// TIA Portal V19 export
FUNCTION_BLOCK "TYPIC_C402_IF_VKL"   // FB112, FBD
TITLE = TYPIC_C402_IF_VKL: Verkeerslicht
{ S7_Optimized_Access := 'TRUE' }
AUTHOR : OCOTECH
FAMILY : Typical
NAME : C402.702
// Logisch Object Besturing: C402.702
// 
// De interne functie verkeerslicht verzorgt de interne besturing, bewaking en fysieke aansturing van een verkeerslicht.
// 
// Het verkeerslicht kan via sturingen (vanuit 3B) of via handmatige bedieningen (aanraakscherm) op volgende standen gezet worden:
//  UIT (gedoofd)
//  ROOD
//  GROEN
//  GEEL KNIPPEREN
// 
// De stand “Geel vast” kan niet via sturing of bediening gekozen worden. De stand “Geel vast” wordt door deze typical altijd automatisch toegepast als overgang naar stand “Rood”.
// stored: MemoryReserve 10, SetENOAutomatically false
   VAR_INPUT
      EXT_AUT { ExternalAccessible := 'False'; ExternalVisible := 'False'; ExternalWritable := 'False'} : Bool;   // Externe (hoofd) beveiliging (1 = OK)
      EXT_HW { ExternalAccessible := 'False'; ExternalVisible := 'False'; ExternalWritable := 'False'} : Bool;   // Sturings hardware (PLC) bewaking (1 = OK)
      HULP_KNIP { ExternalAccessible := 'False'; ExternalVisible := 'False'; ExternalWritable := 'False'} : Bool;   // Knippersignaal, x tijd Hoog, x tijd Laag
      IN_AUT_C402 { ExternalAccessible := 'False'; ExternalVisible := 'False'; ExternalWritable := 'False'} : Bool;   // Beveiligingen: serie geschakelde terugmelding (1 = OK)
      IN_ROOD { ExternalAccessible := 'False'; ExternalVisible := 'False'; ExternalWritable := 'False'} : Bool;   // Terugmelding: rood aan (stroommeting)
      IN_GEEL { ExternalAccessible := 'False'; ExternalVisible := 'False'; ExternalWritable := 'False'} : Bool;   // Terugmelding: geel aan (stroommeting)
      IN_GROE { ExternalAccessible := 'False'; ExternalVisible := 'False'; ExternalWritable := 'False'} : Bool;   // Terugmelding: groen aan (stroommeting)
      CFG_TYD_FB { ExternalAccessible := 'False'; ExternalVisible := 'False'; ExternalWritable := 'False'} : Time;   // Vertragingstijd storing terugmelding
      CFG_GEEL_TYD { ExternalAccessible := 'False'; ExternalVisible := 'False'; ExternalWritable := 'False'} : Time;   // Tijdsduur verkeerslicht geel, vooraleer naar rood
      CFG_SNEL_GEEL_TYD { ExternalAccessible := 'False'; ExternalVisible := 'False'; ExternalWritable := 'False'} : Time;   // Tijdsduur verkeerslicht geel, vooraleer naar rood, bij versneld sluiten
      CFG_TYD_ONHD { ExternalAccessible := 'False'; ExternalVisible := 'False'; ExternalWritable := 'False'} : Time;   // Tijdsduur aansturing lenzen bij automatische onderhoudstesten
   END_VAR
   VAR_OUTPUT
      VAR_IF_VKL { ExternalAccessible := 'False'; ExternalVisible := 'False'; ExternalWritable := 'False'} : "C402_VAR_IF_VKL_TYPIC";   // Struct met alle variabelen naar bovenliggende functies
      OUT_ROOD { ExternalAccessible := 'False'; ExternalVisible := 'False'; ExternalWritable := 'False'} : Bool;   // Aansturing rood
      OUT_GEEL { ExternalAccessible := 'False'; ExternalVisible := 'False'; ExternalWritable := 'False'} : Bool;   // Aansturing geel
      OUT_GROE { ExternalAccessible := 'False'; ExternalVisible := 'False'; ExternalWritable := 'False'} : Bool;   // Aansturing groen
   END_VAR
   VAR_IN_OUT
      STU_IF_VKL : "C402_STU_IF_VKL_TYPIC";   // Struct met alle sturingen naar de functie (IF) in de interne sturing van het verkeerslicht
      STU_AFS_IF_VKL : "C402_STU_AFS_IF_VKL_TYPIC";   // Struct met alle sturingen naar de functie (IF) van de verkeerslichten
   END_VAR
   VAR
      STO { ExternalWritable := 'False'} : Struct   // Storingen
         A001 { ExternalAccessible := 'False'; ExternalVisible := 'False'} : Bool;   // Beveiliging aangesproken
         AT01 { ExternalAccessible := 'False'; ExternalVisible := 'False'} : Bool;   // De rode lens is defect
         AT02 { ExternalAccessible := 'False'; ExternalVisible := 'False'} : Bool;   // De gele lens is defect
         AT03 { ExternalAccessible := 'False'; ExternalVisible := 'False'} : Bool;   // De groene lens is defect
         AT04 { ExternalAccessible := 'False'; ExternalVisible := 'False'} : Bool;   // De stand rood kan niet getoond worden
         AT05 { ExternalAccessible := 'False'; ExternalVisible := 'False'} : Bool;   // De stand geel kan niet getoond worden
         AT06 { ExternalAccessible := 'False'; ExternalVisible := 'False'} : Bool;   // De stand geel knipperen kan niet getoond worden
         AT07 { ExternalAccessible := 'False'; ExternalVisible := 'False'} : Bool;   // De stand groen kan niet getoond worden
      END_STRUCT;
      VAR { ExternalWritable := 'False'} : Struct   // Variabelen
         HAND_ROOD_SWA { ExternalAccessible := 'False'; ExternalVisible := 'False'} : Bool;   // 1 = Rood gewenst, via handbediening
         HAND_KNIP_SWA { ExternalAccessible := 'False'; ExternalVisible := 'False'} : Bool;   // 1 = Geel knipperen gewenst, via handbediening
         HAND_GROE_SWA { ExternalAccessible := 'False'; ExternalVisible := 'False'} : Bool;   // 1 = Groen gewenst, via handbediening
         ROOD_SWA { ExternalAccessible := 'False'; ExternalVisible := 'False'} : Bool;   // 1 = Rood gewenst
         KNIP_SWA { ExternalAccessible := 'False'; ExternalVisible := 'False'} : Bool;   // 1 = Geel knipperen gewenst
         GROEN_SWA { ExternalAccessible := 'False'; ExternalVisible := 'False'} : Bool;   // 1 = Groen gewenst
         ROOD_AAN_SWA { ExternalAccessible := 'False'; ExternalVisible := 'False'} : Bool;   // 1 = Rood gewenst, rode lens aansturen
         GEEL_AAN_SWA { ExternalAccessible := 'False'; ExternalVisible := 'False'} : Bool;   // 1 = Rood gewenst, gele lens aansturen
         GEEL_KNIP { ExternalAccessible := 'False'; ExternalVisible := 'False'} : Bool;   // Knippersignaal voor geel licht 1 = AAN / 0 = UIT
         STO_ROOD_AAN { ExternalAccessible := 'False'; ExternalVisible := 'False'} : Bool;   // 1 = Rode lens defect, geen terugmelding bij aansturen
         STO_ROOD_UIT { ExternalAccessible := 'False'; ExternalVisible := 'False'} : Bool;   // 1 = Rode lens defect, terugmelding aan bij afsturen
         STO_GEEL_AAN { ExternalAccessible := 'False'; ExternalVisible := 'False'} : Bool;   // 1 = Gele lens defect, geen terugmelding bij aansturen
         STO_GEEL_UIT { ExternalAccessible := 'False'; ExternalVisible := 'False'} : Bool;   // 1 = Gele lens defect, terugmelding aan bij afsturen
         STO_GROE_AAN { ExternalAccessible := 'False'; ExternalVisible := 'False'} : Bool;   // 1 = Groene lens defect, geen terugmelding bij aansturen
         STO_GROE_UIT { ExternalAccessible := 'False'; ExternalVisible := 'False'} : Bool;   // 1 = Groene lens defect, terugmelding aan bij afsturen
         ONHD { ExternalAccessible := 'False'; ExternalVisible := 'False'} : Bool;   // 1 = Alle lenzen aansturen ifv onderhoudstesten
         STS_ROOD { ExternalAccessible := 'False'; ExternalVisible := 'False'} : Bool;   // TRUE = Verkeerslicht actueel op rood
         STS_GEEL { ExternalAccessible := 'False'; ExternalVisible := 'False'} : Bool;   // TRUE = Verkeerslicht actueel op geel (vast)
         STS_GROE { ExternalAccessible := 'False'; ExternalVisible := 'False'} : Bool;   // TRUE = Verkeerslicht actueel op groen
         STS_KNIP { ExternalAccessible := 'False'; ExternalVisible := 'False'} : Bool;   // TRUE = Verkeerslicht actueel op knipperen geel
         STS_AAN { ExternalAccessible := 'False'; ExternalVisible := 'False'} : Bool;   // TRUE = Verkeerslicht wordt aangestuurd
         BMO_HAND { ExternalAccessible := 'False'; ExternalVisible := 'False'} : Bool;   // TRUE = Verkeerslicht in hand geschakeld / FALSE = niet in hand
         EXT_AUT { ExternalAccessible := 'False'; ExternalVisible := 'False'} : Bool;   // Externe (hoofd) beveiliging aangesproken
         EXT_HW { ExternalAccessible := 'False'; ExternalVisible := 'False'} : Bool;   // Sturings hardware (PLC) in storing
      END_STRUCT;
   END_VAR
BEGIN

REGION Network 1: START
END_REGION

REGION Network 2: +++ Bepalen bedieningsmode +++
   // Bedieningsmode (Afstand / Hand) bepalen.
END_REGION

REGION Network 3: +++ Bepalen gewenste status +++
   // Gewenste status van het verkeerslicht bepalen (Rood / Geel Knipperen / Groen / Uit).
END_REGION

REGION Network 4: +++ Overgang naar rood +++
   // Als de gewenste stand Rood is, zal er eerst een overgang zijn waarbij het verkeerslicht op geel wordt aangestuurd.
END_REGION

REGION Network 5: +++ Storingen +++
   // Terugmeldingsbewaking van iedere lens.
END_REGION

REGION Network 6: Storing A001: Beveiliging aangesproken
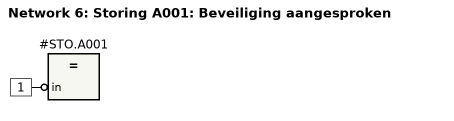
   #STO.A001 := NOT 1;
END_REGION

REGION Network 7: +++ Bepalen actuele status +++
   // Actuele status van het verkeerslicht (Rood / Geel / Geel Knipperen / Groen / Uit).
END_REGION

REGION Network 8: +++ Automatische onderhoudstesten +++
   // Alle lenzen kortstondig en gelijktijdig aansturen ter controle van de goede werking.
END_REGION

REGION Network 9: +++ Aansturing lenzen +++
   // Aansturen van iedere lens (Aan / Uit).
END_REGION

REGION Network 10 (SCL): EINDE
   // Variabelen van intern scada rakvlak naar outputs copieren
   #VAR_IF_VKL.STS_ROOD := #VAR.STS_ROOD;
   #VAR_IF_VKL.STS_GEEL := #VAR.STS_GEEL;
   #VAR_IF_VKL.STS_GROE := #VAR.STS_GROE;
   #VAR_IF_VKL.STS_KNIP := #VAR.STS_KNIP;
   #VAR_IF_VKL.STS_AAN := #VAR.STS_AAN;
   #VAR_IF_VKL.BMO_HAND := #VAR.BMO_HAND;
   #VAR_IF_VKL.EXT_AUT := #VAR.EXT_AUT;
   #VAR_IF_VKL.EXT_HW := #VAR.EXT_HW;
   #VAR_IF_VKL.STO := #STO;
END_REGION
END_FUNCTION_BLOCK
